// SIMATIC S7-200 project (STEP 7-Micro/WIN), CPU 224XP REL 02.01

SYMBOL_TABLE USUARIO1
MARCHA           I0.0
PARO             I0.1
TERMICO          I0.2
MOTOR1           Q0.0
LEDMOTOR1        Q0.1
MOTOR2           Q0.2
LEDMOTOR2        Q0.3
LEDPARO          Q0.4
LEDAVERIA        Q0.5
END_SYMBOL_TABLE

SYMBOL_TABLE Símbolos S7-200
Primer_ciclo_ON  SM0.1    // ON sólo en el primer ciclo
END_SYMBOL_TABLE

ORGANIZATION_BLOCK PRINCIPAL:OB1
TITLE=COMENTARIOS DEL PROGRAMA
BEGIN
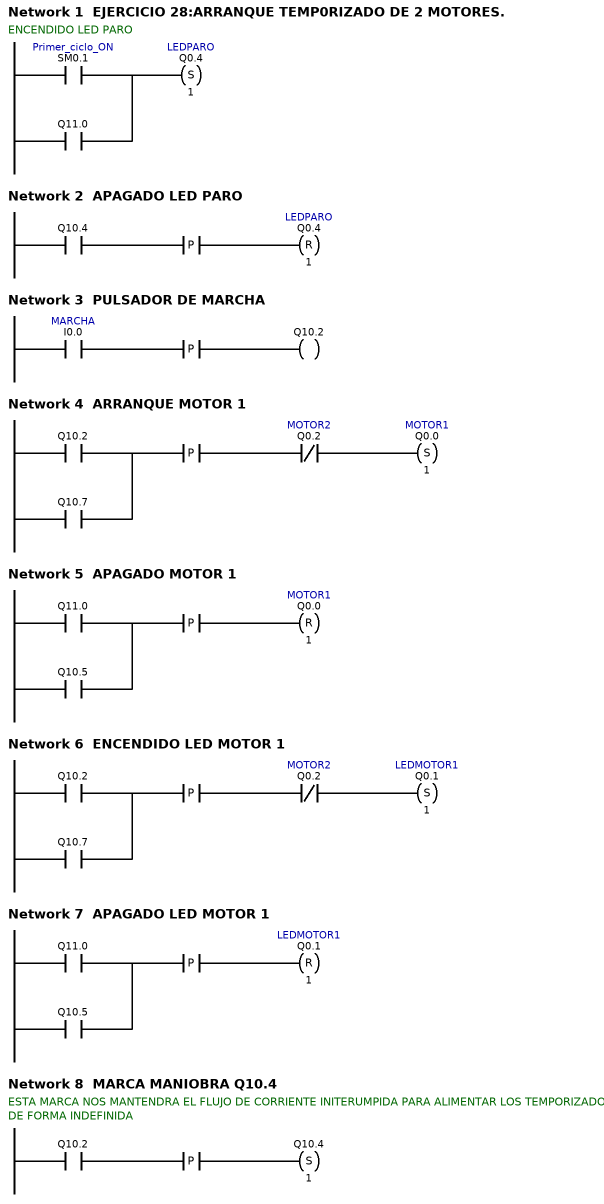
Network 1 // EJERCICIO 28:ARRANQUE TEMP0RIZADO DE 2 MOTORES.
// ENCENDIDO LED PARO
LD     Primer_ciclo_ON:SM0.1
O      Q11.0
S      LEDPARO:Q0.4, 1
Network 2 // APAGADO LED PARO
LD     Q10.4
EU
R      LEDPARO:Q0.4, 1
Network 3 // PULSADOR DE MARCHA
LD     MARCHA:I0.0
EU
=      Q10.2
Network 4 // ARRANQUE MOTOR 1 
LD     Q10.2
O      Q10.7
EU
AN     MOTOR2:Q0.2
S      MOTOR1:Q0.0, 1
Network 5 // APAGADO MOTOR 1 
LD     Q11.0
O      Q10.5
EU
R      MOTOR1:Q0.0, 1
Network 6 // ENCENDIDO LED MOTOR 1 
LD     Q10.2
O      Q10.7
EU
AN     MOTOR2:Q0.2
S      LEDMOTOR1:Q0.1, 1
Network 7 // APAGADO LED MOTOR 1 
LD     Q11.0
O      Q10.5
EU
R      LEDMOTOR1:Q0.1, 1
Network 8 // MARCA MANIOBRA Q10.4
// ESTA MARCA NOS MANTENDRA EL FLUJO DE CORRIENTE INITERUMPIDA PARA ALIMENTAR LOS TEMPORIZADORES Y ASI CONSEGUIR INTERMITENCIA , POR SUPUESTO QUE UNO DESCONECTA AL OTRO DE FORMA INDEFINIDA
LD     Q10.2
EU
S      Q10.4, 1
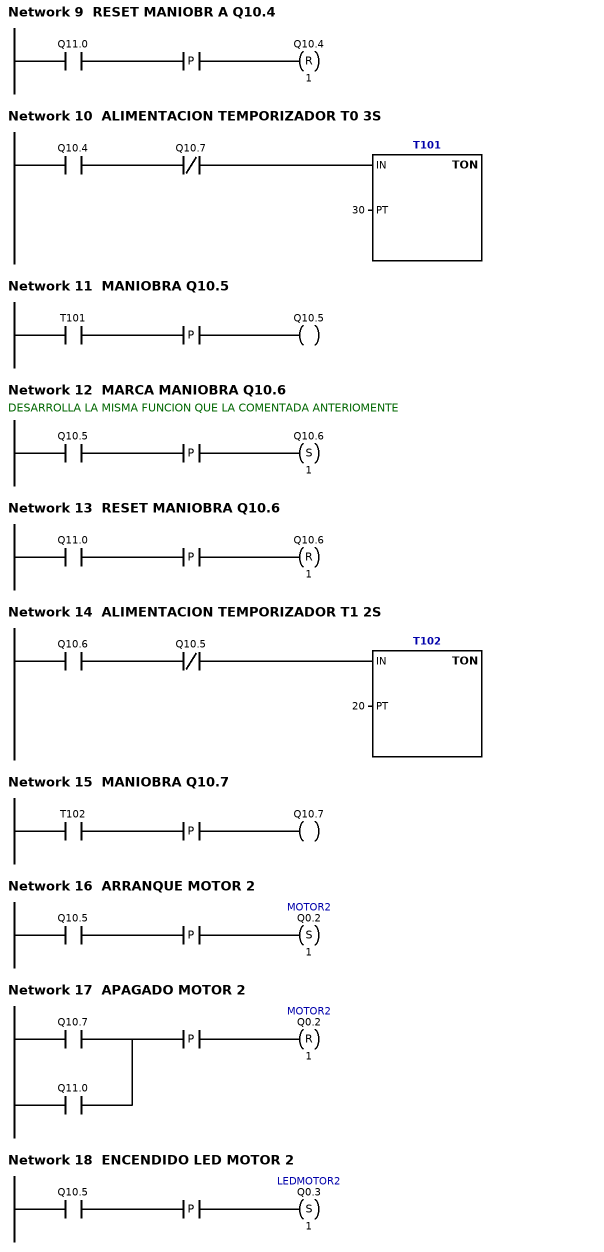
Network 9 // RESET MANIOBR A Q10.4
LD     Q11.0
EU
R      Q10.4, 1
Network 10 // ALIMENTACION TEMPORIZADOR T0 3S
LD     Q10.4
AN     Q10.7
TON    T101, 30
Network 11 // MANIOBRA Q10.5
LD     T101
EU
=      Q10.5
Network 12 // MARCA MANIOBRA Q10.6
// DESARROLLA LA MISMA FUNCION QUE LA COMENTADA ANTERIOMENTE
LD     Q10.5
EU
S      Q10.6, 1
Network 13 // RESET MANIOBRA Q10.6
LD     Q11.0
EU
R      Q10.6, 1
Network 14 // ALIMENTACION TEMPORIZADOR T1 2S
LD     Q10.6
AN     Q10.5
TON    T102, 20
Network 15 // MANIOBRA Q10.7
LD     T102
EU
=      Q10.7
Network 16 // ARRANQUE MOTOR 2
LD     Q10.5
EU
S      MOTOR2:Q0.2, 1
Network 17 // APAGADO MOTOR 2 
LD     Q10.7
O      Q11.0
EU
R      MOTOR2:Q0.2, 1
Network 18 // ENCENDIDO LED MOTOR 2 
LD     Q10.5
EU
S      LEDMOTOR2:Q0.3, 1
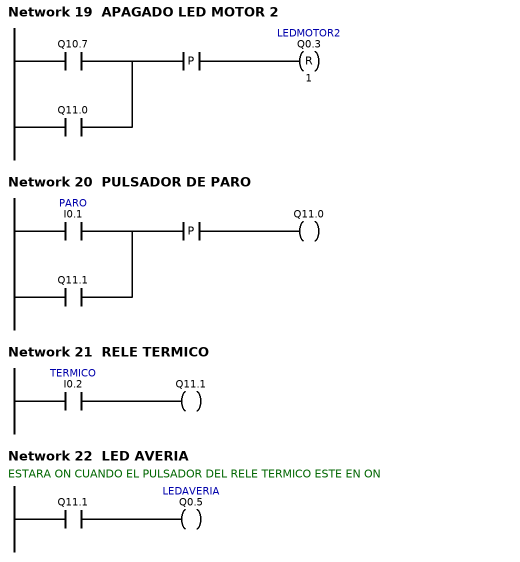
Network 19 // APAGADO LED MOTOR 2 
LD     Q10.7
O      Q11.0
EU
R      LEDMOTOR2:Q0.3, 1
Network 20 // PULSADOR DE PARO 
LD     PARO:I0.1
O      Q11.1
EU
=      Q11.0
Network 21 // RELE TERMICO
LD     TERMICO:I0.2
=      Q11.1
Network 22 // LED AVERIA
// ESTARA ON CUANDO EL PULSADOR DEL RELE TERMICO ESTE EN ON 
LD     Q11.1
=      LEDAVERIA:Q0.5
END_ORGANIZATION_BLOCK
